FUNCTION_BLOCK TelemetryPack (* Telemetry_CAT helper: packs the MQTT_CONNECTION status scalars into the TelemetryHealth struct (scalar in + ST member access -> whole-struct out — no struct-member connections, which EAE rejects) *)
  (* Standard: 61499-2 *)
  (* Version 0.1, 6/22/2026, easensoy, WMG, IsConnected/ReturnCode/Status/NetworkState/SecurityState/ProtocolState -> Health:TelemetryHealth *)
  PACKAGE Main;
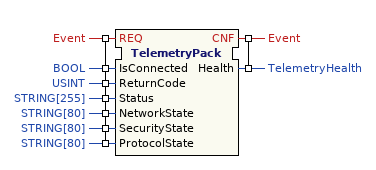
  EVENT_INPUT
    REQ WITH IsConnected, ReturnCode, Status, NetworkState, SecurityState, ProtocolState; (* Pack request *)
  END_EVENT
  EVENT_OUTPUT
    CNF WITH Health; (* Pack confirm *)
  END_EVENT
  VAR_INPUT
    IsConnected : BOOL;
    ReturnCode : USINT;
    Status : STRING[255];
    NetworkState : STRING[80];
    SecurityState : STRING[80];
    ProtocolState : STRING[80];
  END_VAR
  VAR_OUTPUT
    Health : TelemetryHealth; (* Resource telemetry connection health *)
  END_VAR
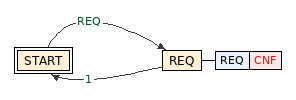
  EC_STATES
    START; (* Initial State *)
    REQ : REQ -> CNF; (* Pack *)
  END_STATES
  EC_TRANSITIONS
    START TO REQ := REQ;
    REQ TO START := 1;
  END_TRANSITIONS
  ALGORITHM REQ IN ST: (* Copy each status scalar into the Health struct *)
Health.IsConnected := IsConnected;
Health.ReturnCode := ReturnCode;
Health.Status := Status;
Health.NetworkState := NetworkState;
Health.SecurityState := SecurityState;
Health.ProtocolState := ProtocolState;
  END_ALGORITHM
END_FUNCTION_BLOCK
